FUNCTION_BLOCK MUX_BYTE (* See MUX_ANY *)
  (* Standard: 61131-3 *)
  (* Version 0.0, 2004-12-15, JHC, Rockwell Automation, Converted from SRC format. *)
  (* Compiler header: package fb.rt.plc.select; *)
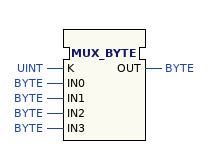
  VAR_INPUT
    K : UINT;
    IN0 : BYTE;
    IN1 : BYTE;
    IN2 : BYTE;
    IN3 : BYTE;
  END_VAR
  VAR_OUTPUT
    OUT : BYTE;
  END_VAR
END_FUNCTION_BLOCK
